      back_feature = get_feature_plane_xz(b_p1,b_p2,b_p3)
      wv_wp1 = pose_trans(wv_wp1,p[0,0,0,0,0,d2r(-90)])
      wv_wp1 = feature_offset(wv_wp1,p[0,offset_2f_k/1000,0,0,0,0],back_feature)
      wv_wp1 = pose_add(wv_wp1,p[0,0,offset_2f_z/1000,0,0,0])
      # wv_wp1 = pose_add(wv_wp1,p[offset_2f_k/1000,0,0,0,0,0])
    end
      # wv_wp2 = pose_add(wv_wp2,p[offset_2f_k/1000,0,0,0,0,0])
      wv_wp2 = feature_offset(wv_wp2,p[0,offset_2f_k/1000,0,0,0,0],back_feature)
      wv_wp2 = pose_add(wv_wp2,p[0,0,offset_2f_z/1000,0,0,0])
      wv_wp2 = p[wv_wp2[0],wv_wp2[1],wv_wp2[2],wv_wp1[3],wv_wp1[4],wv_wp1[5]]

      wv_wp3_p = feature_offset(wv_wp3[0],p[0,offset_2f_k/1000,0,0,0,0],back_feature)
      wv_wp3_p = pose_add(wv_wp3_p,p[0,0,offset_2f_z/1000,0,0,0])
      wv_wp3_p = p[wv_wp3_p[0],wv_wp3_p[1],wv_wp3_p[2],wv_wp1[3],wv_wp1[4],wv_wp1[5]]
      wv_wp4[0] = p[wv_wp3_p[0],wv_wp3_p[1],wv_wp3_p[2],wv_wp1[3],wv_wp1[4],wv_wp1[5]]

      wv_wp3_p = feature_offset(wv_wp3[1],p[0,offset_2f_k/1000,0,0,0,0],back_feature)
      wv_wp3_p = pose_add(wv_wp3_p,p[0,0,offset_2f_z/1000,0,0,0])
      wv_wp3_p = p[wv_wp3_p[0],wv_wp3_p[1],wv_wp3_p[2],wv_wp1[3],wv_wp1[4],wv_wp1[5]]
      wv_wp4[1] = p[wv_wp3_p[0],wv_wp3_p[1],wv_wp3_p[2],wv_wp1[3],wv_wp1[4],wv_wp1[5]]

      wv_wp3_p = feature_offset(wv_wp3[2],p[0,offset_2f_k/1000,0,0,0,0],back_feature)
      wv_wp3_p = pose_add(wv_wp3_p,p[0,0,offset_2f_z/1000,0,0,0])
      wv_wp3_p = p[wv_wp3_p[0],wv_wp3_p[1],wv_wp3_p[2],wv_wp1[3],wv_wp1[4],wv_wp1[5]]
      wv_wp4[2] = p[wv_wp3_p[0],wv_wp3_p[1],wv_wp3_p[2],wv_wp1[3],wv_wp1[4],wv_wp1[5]]
  end
  if(ext_fun[2]==1 and par_2f==False):
    #squash
    w_voltage = ext_fun[3]
    w_current = ext_fun[4]
    set_current_voltage(w_current,w_voltage)
    global cir_speed_org_bak = wv_weldpar[1]
    global wving_amplitude_bak = wv_weldpar[4]
    wv_weldpar[1] = ext_fun[6]
    wv_weldpar[4] = ext_fun[5]
  end
  if(par_2f):
    global wv_system_speed = calculate_2f(wv_weldpar[4],wv_wp1,wv_wp2,wv_weldpar[1],wv_weldpar[3],wving_delay,wving_crater,wv_weldpar[6])
  else:
    global wv_system_speed = calculate_3f(wv_weldpar[4],wv_wp1,wv_wp2,wv_weldpar[1],wv_weldpar[3],wving_delay)
    x_radius = x_radius / 1000
  end
  global wv_set_speed = wv_system_speed
  ratio_t=0
  # mm -> m
  global y_radius = y_radius / 1000
  global y_radius_bak = y_radius
  #init for thread
  global ext_stick = 0
  global th_arc_sen=Arc_sen
  global th_wv_gap=wv_gap
  global th_tilt_deg=tilt_deg

  global last_tilt_deg =th_tilt_deg
  global last_wv_wp1 = wv_wp1
  global last_wv_line = wv_Line_Feature2
  global th_wving_crater=wving_crater
  global last_z_bottom = z_bottom
  global th_par_2f = par_2f
  global th_cir_speed_org=wv_weldpar[1]
  global th_wv_wp1 = wv_wp1
  global th_wv_wp2 = wv_wp2
  global th_wv_wp3 = wv_wp3[0]
  global th_wv_weldpar=wv_weldpar
  global th_wving_delay=wving_delay
  global th_z_param=z_param
  global th_wv_seq = wv_seq
  global th_wv_feature=wv_feature
  global th_dir = dir

  # if want to use approach position
  if(wv_seq[0] ==0 or wv_seq[0] == 1):
    global get_angle_rx = welding_angle_cal_2f(wv_wp1[1],tilt_deg,vir_v,cal_off_ang_rx)
    global get_angle_ry = welding_angle_cal_3f(wv_wp1[2],tilt_deg,z_bottom,cal_off_ang_ry)

    target_p = feature_offset(wv_wp1,p[0,0,0,d2r(tilt_deg[0] + get_angle_rx),d2r(tilt_deg[1] + get_angle_ry),d2r(tilt_deg[2])],wv_Line_Feature2)

    if(wv_weldpar[2]==1):
      target_p_appr = feature_offset(target_p,p[0,0,-0.02,0,0,0],wv_Line_Feature2)
      movel(target_p_appr,a=0.5,v=0.125)
    end
    movel(target_p,a=0.5,v=0.125)
  end

  CThread = run CalThread()
  DThread = run diff_Thread()
  TThread = run thread_timer()
  AThread = run Arc_Thread()
  TTRRhread = run thread_dist_rec()

  global timer_counting=True
  global program_weld_on = True

  if(a9_wv_weldingon==True):
    while(welding_off_t==55):
      sync()
    end
    if(wving_crater[2]>0):
      set_current_voltage(wving_crater[0],wving_crater[1])
    end
    if(welding_off_t != 1):
      write_welder(0,True)
      while(get_wcr==False):
        if(weld_onoff==False):
          write_welder(0,True)
        end
        sync()
      end
      if(wving_crater[2]>0):
        #Crater Begin option
        write_output_float_register(1,1)
        sleep(wving_crater[2])
        set_current_voltage(ext_fun[1],ext_fun[0])
      end
    end
  end
  start_gas_time = 0

  background_cal=1
  background_ready=0
  FT_trig=True

  timer_1_is_counting = True

  while((ratio_t < 1) or current_list==0 or current_list==1):
    if(ratio_t>=1 and current_list!=2):
      if (gap_check):
        gap_check = True
        wv_gap[0]=1
        th_wv_gap[0]=1
        gap_check= False
      end
      ratio_t=0
      if(current_list==0):
        wving_amp_bak = wv_weldpar[4]
        wv_weldpar[4] = wv_weldpar[4] * 1
        th_wv_weldpar[4] = wv_weldpar[4]
        circle_speed_bak = wv_weldpar[1]
        wv_weldpar[1]= wv_weldpar[1]*0.7
        th_wv_weldpar[1]= wv_weldpar[1]
      elif(current_list==1):
        wv_weldpar[4] = wving_amp_bak
        th_wv_weldpar[4] = wv_weldpar[4]
        wv_weldpar[1] = circle_speed_bak
        th_wv_weldpar[1]= wv_weldpar[1]
      end
      wv_wp1=wv_wp4[current_list]
      wv_wp2=wv_wp4[current_list+1]
      global th_wv_wp1 = wv_wp4[current_list]
      global th_wv_wp2 = wv_wp4[current_list+1]
      global th_wv_wp3 = wv_wp4[current_list+1]
      wv_system_speed_bak = wv_system_speed
      if(par_2f):
        global wv_system_speed = calculate_2f(wv_weldpar[4],wv_wp4[current_list],wv_wp4[current_list+1],wv_weldpar[1],wv_weldpar[3],wving_delay,wving_crater)
        global y_radius = y_radius / 1000
        global y_radius_bak = y_radius
      else:
        global wv_system_speed = calculate_3f(wv_weldpar[4],wv_wp4[current_list],wv_wp4[current_list+1],wv_weldpar[1],wv_weldpar[3],wving_delay)
        x_radius = x_radius / 1000
      end
      wv_system_speed = wv_system_speed_bak
      current_list=current_list+1
    end

    if( (norm(tri_count)>=2 and par_2f==False or FT_trig==True) or (norm(tri_count)>=4 and par_2f==True or FT_trig==True)   ):
      FT_trig = False
      while(background_ready==0):
        sync()
      end
      tri_count = 0
      background_ready = 0
      global move_p = background_pose
      wv_wp2 = th_wv_wp2
      if(par_2f):
        background_cal=1
      else:
        background_cal=1
      end
      global a_val = 3
      if(a_val >= 30):
        write_port_register(142,112)
        sleep(0.5)
        halt
      end
    end

    if(wv_weldpar[5] ==1):
        if( (sin_dir==1 and wving_delay[0]==0) or (sin_dir==-1 and wving_delay[2]==0)):
         tri_count = tri_count + 1
        end
        # write_output_float_register(24,tri_count)
        global target_p = move_p[tri_count]
        target_p=p[target_p[0],target_p[1],target_p[2],target_p[3],target_p[4],target_p[5]]
        tri_count = tri_count + 1
    elif(wv_weldpar[5] ==2):
      if( (tri_count==1 and sin_dir==1 and wving_delay[0]==0) or (tri_count==1 and sin_dir==-1 and wving_delay[2]==0)):
       tri_count = tri_count + 1
      end
      # write_output_float_register(24,tri_count)
      global target_p = move_p[tri_count]
      target_p=p[target_p[0],target_p[1],target_p[2],target_p[3],target_p[4],target_p[5]]
      tri_count = tri_count + 1
    else:
      popup("Please insert 0 - sin or 1 - triangle")
    end

    if(target_p == p[0,0,0,0,0,0]):
      target_p = get_actual_tcp_pose()
    end
    # write_output_float_register(23,sin_dir)
    ARC_T_ONOFF = True
    ARC_T_s_pose = get_actual_tcp_pose()
    ARC_T_e_pose = target_p
    if((norm(tri_count)== 2) and wving_delay[1]>0 and par_2f):
      # DOWN
      movel(target_p,a=a_val,v=wv_system_speed/1000)
      sleep(wving_delay[1])
    elif((norm(tri_count)== 4) and wving_delay[3]>0 and par_2f):
      #UP
      movel(target_p,a=a_val,v=wv_system_speed/1000)
      sleep(wving_delay[3])
    elif((norm(tri_count)== 2) and sin_dir==1 and wving_delay[1]>0 and par_2f == False):
      movel(target_p,a=a_val,v=wv_system_speed/1000)
      sleep(wving_delay[1])
    elif((norm(tri_count)== 2) and sin_dir==-1 and wving_delay[3]>0 and par_2f == False):
      movel(target_p,a=a_val,v=wv_system_speed/1000)
      sleep(wving_delay[3])
    elif((norm(tri_count)== 1) and wving_delay[0]>0 and par_2f):
      movel(target_p,a=a_val,v=wv_system_speed/1000)
      sleep(wving_delay[0])
    elif((norm(tri_count)== 3) and wving_delay[2]>0 and par_2f):
      movel(target_p,a=a_val,v=wv_system_speed/1000)
      sleep(wving_delay[2])
    else:
      movel(target_p,a=a_val,v=wv_system_speed/1000)
    end
    global last_pose = target_p
  end

  timer_1_is_counting = False
  welding_program = True
  if(a9_wv_weldingon == True and wving_crater[5]!=0):
    #crater end option
    set_current_voltage(wving_crater[3],wving_crater[4])
    sleep(wving_crater[5])
    program_weld_on = False
    set_current_voltage(ext_fun[1],ext_fun[0])
    if(isHicomm):
      write_port_register(202,0)
      write_port_register(149,0)
    else:
      set_standard_digital_out(0,False)
    end
    while(get_wcr==True):
      if(weld_onoff==True):
        if(isHicomm):
          write_port_register(202,0)
          write_port_register(149,0)
        else:
          set_standard_digital_out(0,False)
        end
      end
      sync()
    end
  end

  kill CThread
  kill DThread
  kill TThread
  kill AThread
  kill TTRRhread
  ARC_T_ONOFF=False
  timer_counting = False
  wcr_counter = 0
  wcr_counting = False
  get_wcr = False
  welding_off_t = 0
  plus_alpha_x = 0
  plus_alpha_z = 0

  if(wv_seq[0] == 0 or wv_seq[0] == 3):
    if(a9_wv_weldingon==True):
      program_weld_on = False
      if(isHicomm):
        write_port_register(202,0)
        write_port_register(149,0)
      else:
        set_standard_digital_out(0,False)
      end
      if(wv_weldpar[2]==1):
        target_pos = feature_offset(get_actual_tcp_pose(),p[0,0,-0.01,0,0,0],wv_Line_Feature2)
        movel(target_pos,0.5,0.01)
      end
    end
  end
  background_pose = [dumy_p,dumy_p,dumy_p,dumy_p]
  move_p = background_pose
  return sin_dir
end
